FUNCTION_BLOCK Bank (* Composite Function Block Type *)
  (* Standard: 61499-2 *)
  (* Version 0.0, 02/03/2026, template *)
  PACKAGE Hidryco.HidrycoLib;
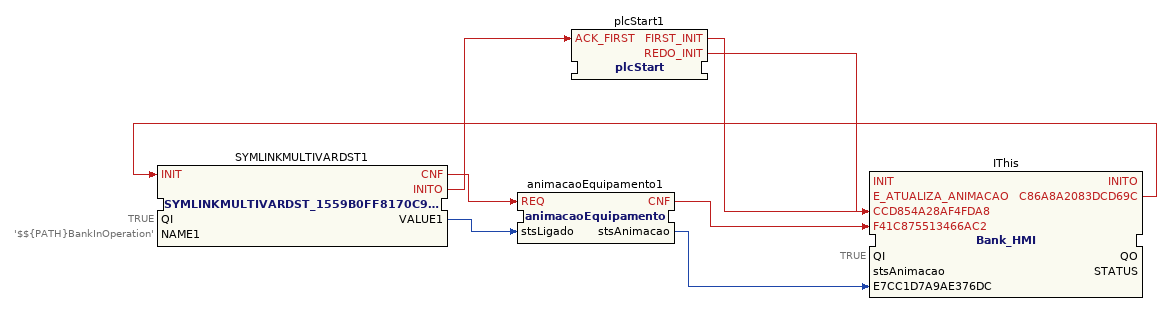
  FBS
    SYMLINKMULTIVARDST1 : SYMLINKMULTIVARDST_1559B0FF8170C9BA0(QI := TRUE, NAME1 := '$${PATH}BankInOperation'); {SET_ATTRIBUTE(Configuration.GenericFBType.InterfaceParams, Runtime.System#I:=1;VALUE${I$}:BOOL)}
    animacaoEquipamento1 : animacaoEquipamento;
    IThis : Bank_HMI(QI := TRUE);
    plcStart1 : plcStart;
  END_FBS
  EVENT_CONNECTIONS
    SYMLINKMULTIVARDST1.CNF TO animacaoEquipamento1.REQ;
    plcStart1.FIRST_INIT TO IThis.CCD854A28AF4FDA8;
    plcStart1.REDO_INIT TO IThis.CCD854A28AF4FDA8;
    animacaoEquipamento1.CNF TO IThis.F41C875513466AC2;
    IThis.C86A8A2083DCD69C TO SYMLINKMULTIVARDST1.INIT;
    SYMLINKMULTIVARDST1.INITO TO plcStart1.ACK_FIRST;
  END_CONNECTIONS
  DATA_CONNECTIONS
    SYMLINKMULTIVARDST1.VALUE1 TO animacaoEquipamento1.stsLigado;
    animacaoEquipamento1.stsAnimacao TO IThis.E7CC1D7A9AE376DC;
  END_CONNECTIONS
END_FUNCTION_BLOCK
